PROGRAM prgAfterStationScan
VAR
END_VAR

//theme:ldUT4FLxql4
//call at the end of scan of stations..
//..for data to be processed after all values of a station
actAnyAlarmsGlobal();
actAnyWarningGlobal();

ACTION actAnyAlarmsGlobal:
//call for end of scan
//if any station has fault state, then set logic for all stations...
//writes to data multiple times due to manipulation of scan
IF 
	GlobalMessages.gMsgS1Stat.IsAlarm OR 
	GlobalMessages.gMsgS2Stat.IsAlarm OR 
	GlobalMessages.gMsgS3Stat.IsAlarm OR 
	GlobalMessages.gMsgS4Stat.IsAlarm OR 
	GlobalMessages.gMsgS5Stat.IsAlarm OR 
	GlobalMessages.gMsgS6Stat.IsAlarm OR
	GlobalMessages.gMsgMcStat.IsAlarm
THEN
	S1_Global.hmiHeader.AnyStationFaultHeaderActive := System.OneSecond;
	S2_Global.hmiHeader.AnyStationFaultHeaderActive := System.OneSecond;
	S3_Global.hmiHeader.AnyStationFaultHeaderActive := System.OneSecond;
	S4_Global.hmiHeader.AnyStationFaultHeaderActive := System.OneSecond;
	S5_Global.hmiHeader.AnyStationFaultHeaderActive := System.OneSecond;
	S6_Global.hmiHeader.AnyStationFaultHeaderActive := System.OneSecond;
	
	S1_Global.hmiHeader.AnyStationFaultColour		:= HMIColour.colourRed;
	S2_Global.hmiHeader.AnyStationFaultColour		:= HMIColour.colourRed;
	S3_Global.hmiHeader.AnyStationFaultColour		:= HMIColour.colourRed;
	S4_Global.hmiHeader.AnyStationFaultColour		:= HMIColour.colourRed;
	S5_Global.hmiHeader.AnyStationFaultColour		:= HMIColour.colourRed;
	S6_Global.hmiHeader.AnyStationFaultColour		:= HMIColour.colourRed;
	
	S1_Global.hmiHeader.isAnyFaultState				:= TRUE;
	S2_Global.hmiHeader.isAnyFaultState				:= TRUE;
	S3_Global.hmiHeader.isAnyFaultState				:= TRUE;
	S4_Global.hmiHeader.isAnyFaultState				:= TRUE;
	S5_Global.hmiHeader.isAnyFaultState				:= TRUE;
	S6_Global.hmiHeader.isAnyFaultState				:= TRUE;
	
ELSE
	S1_Global.hmiHeader.AnyStationFaultHeaderActive := FALSE;
	S2_Global.hmiHeader.AnyStationFaultHeaderActive := FALSE;
	S3_Global.hmiHeader.AnyStationFaultHeaderActive := FALSE;
	S4_Global.hmiHeader.AnyStationFaultHeaderActive := FALSE;
	S5_Global.hmiHeader.AnyStationFaultHeaderActive := FALSE;
	S6_Global.hmiHeader.AnyStationFaultHeaderActive := FALSE;

	S1_Global.hmiHeader.AnyStationFaultColour		:= HMIColour.colourBlue;
	S2_Global.hmiHeader.AnyStationFaultColour		:= HMIColour.colourBlue;
	S3_Global.hmiHeader.AnyStationFaultColour		:= HMIColour.colourBlue;
	S4_Global.hmiHeader.AnyStationFaultColour		:= HMIColour.colourBlue;
	S5_Global.hmiHeader.AnyStationFaultColour		:= HMIColour.colourBlue;
	S6_Global.hmiHeader.AnyStationFaultColour		:= HMIColour.colourBlue;

	S1_Global.hmiHeader.isAnyFaultState				:= FALSE;
	S2_Global.hmiHeader.isAnyFaultState				:= FALSE;
	S3_Global.hmiHeader.isAnyFaultState				:= FALSE;
	S4_Global.hmiHeader.isAnyFaultState				:= FALSE;
	S5_Global.hmiHeader.isAnyFaultState				:= FALSE;
	S6_Global.hmiHeader.isAnyFaultState				:= FALSE;	
END_IF

	//set indicators to 0
	S1_Global.hmiHeader.AnyStationFaultHeader := 0;
	S2_Global.hmiHeader.AnyStationFaultHeader := 0;
	S3_Global.hmiHeader.AnyStationFaultHeader := 0;
	S4_Global.hmiHeader.AnyStationFaultHeader := 0;
	S5_Global.hmiHeader.AnyStationFaultHeader := 0;
	S6_Global.hmiHeader.AnyStationFaultHeader := 0;

//write station 1 is in fault
IF 	S1_Global.hmiHeader.isFaultState THEN
	S1_Global.hmiHeader.AnyStationFaultHeader := 1;
	S2_Global.hmiHeader.AnyStationFaultHeader := 1;
	S3_Global.hmiHeader.AnyStationFaultHeader := 1;
	S4_Global.hmiHeader.AnyStationFaultHeader := 1;
	S5_Global.hmiHeader.AnyStationFaultHeader := 1;
	S6_Global.hmiHeader.AnyStationFaultHeader := 1;
END_IF

//write station 2 is in fault
IF 	S2_Global.hmiHeader.isFaultState THEN
	S1_Global.hmiHeader.AnyStationFaultHeader := 2;
	S2_Global.hmiHeader.AnyStationFaultHeader := 2;
	S3_Global.hmiHeader.AnyStationFaultHeader := 2;
	S4_Global.hmiHeader.AnyStationFaultHeader := 2;
	S5_Global.hmiHeader.AnyStationFaultHeader := 2;
	S6_Global.hmiHeader.AnyStationFaultHeader := 2;
END_IF

//write station 3 is in fault
IF 	S3_Global.hmiHeader.isFaultState THEN
	S1_Global.hmiHeader.AnyStationFaultHeader := 3;
	S2_Global.hmiHeader.AnyStationFaultHeader := 3;
	S3_Global.hmiHeader.AnyStationFaultHeader := 3;
	S4_Global.hmiHeader.AnyStationFaultHeader := 3;
	S5_Global.hmiHeader.AnyStationFaultHeader := 3;
	S6_Global.hmiHeader.AnyStationFaultHeader := 3;
END_IF

//write station 4 is in fault
IF 	S4_Global.hmiHeader.isFaultState THEN
	S1_Global.hmiHeader.AnyStationFaultHeader := 4;
	S2_Global.hmiHeader.AnyStationFaultHeader := 4;
	S3_Global.hmiHeader.AnyStationFaultHeader := 4;
	S4_Global.hmiHeader.AnyStationFaultHeader := 4;
	S5_Global.hmiHeader.AnyStationFaultHeader := 4;
	S6_Global.hmiHeader.AnyStationFaultHeader := 4;
END_IF

//write station 5 is in fault
IF 	S5_Global.hmiHeader.isFaultState THEN
	S1_Global.hmiHeader.AnyStationFaultHeader := 5;
	S2_Global.hmiHeader.AnyStationFaultHeader := 5;
	S3_Global.hmiHeader.AnyStationFaultHeader := 5;
	S4_Global.hmiHeader.AnyStationFaultHeader := 5;
	S5_Global.hmiHeader.AnyStationFaultHeader := 5;
	S6_Global.hmiHeader.AnyStationFaultHeader := 5;
END_IF

//write station 6 is in fault
IF 	S6_Global.hmiHeader.isFaultState THEN
	S1_Global.hmiHeader.AnyStationFaultHeader := 6;
	S2_Global.hmiHeader.AnyStationFaultHeader := 6;
	S3_Global.hmiHeader.AnyStationFaultHeader := 6;
	S4_Global.hmiHeader.AnyStationFaultHeader := 6;
	S5_Global.hmiHeader.AnyStationFaultHeader := 6;
	S6_Global.hmiHeader.AnyStationFaultHeader := 6;
END_IF

//..so it appears in all usage of the HMI for a given station

//add for base station header
IF GlobalMessages.gMsgMcStat.IsAlarm THEN
	//set special case for base machine
	S1_Global.hmiHeader.AnyStationFaultHeader := 99;
	S2_Global.hmiHeader.AnyStationFaultHeader := 99;
	S3_Global.hmiHeader.AnyStationFaultHeader := 99;
	S4_Global.hmiHeader.AnyStationFaultHeader := 99;
	S5_Global.hmiHeader.AnyStationFaultHeader := 99;
	S6_Global.hmiHeader.AnyStationFaultHeader := 99;
	
	S1_Global.hmiHeader.isFaultState := TRUE;
	S2_Global.hmiHeader.isFaultState := TRUE;
	S3_Global.hmiHeader.isFaultState := TRUE;
	S4_Global.hmiHeader.isFaultState := TRUE;
	S5_Global.hmiHeader.isFaultState := TRUE;
	S6_Global.hmiHeader.isFaultState := TRUE;
	
	S1_Global.hmiHeader.FaultStateHeader := 1;
	S2_Global.hmiHeader.FaultStateHeader := 1;
	S3_Global.hmiHeader.FaultStateHeader := 1;
	S4_Global.hmiHeader.FaultStateHeader := 1;
	S5_Global.hmiHeader.FaultStateHeader := 1;
	S6_Global.hmiHeader.FaultStateHeader := 1;
END_IF
END_ACTION

ACTION actAnyWarningGlobal:
//call for end of scan
//if any station has Warning state, then set logic for all stations...
//writes to data multiple times due to manipulation of scan
IF 
	GlobalMessages.gMsgS1Stat.IsWarning OR 
	GlobalMessages.gMsgS2Stat.IsWarning OR 
	GlobalMessages.gMsgS3Stat.IsWarning OR 
	GlobalMessages.gMsgS4Stat.IsWarning OR 
	GlobalMessages.gMsgS5Stat.IsWarning OR 
	GlobalMessages.gMsgS6Stat.IsWarning OR
	GlobalMessages.gMsgMcStat.IsWarning
THEN
	S1_Global.hmiHeader.AnyStationWarningHeaderActive := System.OneSecond;
	S2_Global.hmiHeader.AnyStationWarningHeaderActive := System.OneSecond;
	S3_Global.hmiHeader.AnyStationWarningHeaderActive := System.OneSecond;
	S4_Global.hmiHeader.AnyStationWarningHeaderActive := System.OneSecond;
	S5_Global.hmiHeader.AnyStationWarningHeaderActive := System.OneSecond;
	S6_Global.hmiHeader.AnyStationWarningHeaderActive := System.OneSecond;
	
	S1_Global.hmiHeader.AnyStationWarningColour		:= HMIColour.colourYellow;
	S2_Global.hmiHeader.AnyStationWarningColour		:= HMIColour.colourYellow;
	S3_Global.hmiHeader.AnyStationWarningColour		:= HMIColour.colourYellow;
	S4_Global.hmiHeader.AnyStationWarningColour		:= HMIColour.colourYellow;
	S5_Global.hmiHeader.AnyStationWarningColour		:= HMIColour.colourYellow;
	S6_Global.hmiHeader.AnyStationWarningColour		:= HMIColour.colourYellow;
	
	S1_Global.hmiHeader.isAnyWarningState				:= TRUE;
	S2_Global.hmiHeader.isAnyWarningState				:= TRUE;
	S3_Global.hmiHeader.isAnyWarningState				:= TRUE;
	S4_Global.hmiHeader.isAnyWarningState				:= TRUE;
	S5_Global.hmiHeader.isAnyWarningState				:= TRUE;
	S6_Global.hmiHeader.isAnyWarningState				:= TRUE;
	
ELSE
	S1_Global.hmiHeader.AnyStationWarningHeaderActive := FALSE;
	S2_Global.hmiHeader.AnyStationWarningHeaderActive := FALSE;
	S3_Global.hmiHeader.AnyStationWarningHeaderActive := FALSE;
	S4_Global.hmiHeader.AnyStationWarningHeaderActive := FALSE;
	S5_Global.hmiHeader.AnyStationWarningHeaderActive := FALSE;
	S6_Global.hmiHeader.AnyStationWarningHeaderActive := FALSE;

	S1_Global.hmiHeader.AnyStationWarningColour		:= HMIColour.colourBlue;
	S2_Global.hmiHeader.AnyStationWarningColour		:= HMIColour.colourBlue;
	S3_Global.hmiHeader.AnyStationWarningColour		:= HMIColour.colourBlue;
	S4_Global.hmiHeader.AnyStationWarningColour		:= HMIColour.colourBlue;
	S5_Global.hmiHeader.AnyStationWarningColour		:= HMIColour.colourBlue;
	S6_Global.hmiHeader.AnyStationWarningColour		:= HMIColour.colourBlue;

	S1_Global.hmiHeader.isAnyWarningState				:= FALSE;
	S2_Global.hmiHeader.isAnyWarningState				:= FALSE;
	S3_Global.hmiHeader.isAnyWarningState				:= FALSE;
	S4_Global.hmiHeader.isAnyWarningState				:= FALSE;
	S5_Global.hmiHeader.isAnyWarningState				:= FALSE;
	S6_Global.hmiHeader.isAnyWarningState				:= FALSE;	
END_IF

	//set indicators to 0
	S1_Global.hmiHeader.AnyStationWarningHeader := 0;
	S2_Global.hmiHeader.AnyStationWarningHeader := 0;
	S3_Global.hmiHeader.AnyStationWarningHeader := 0;
	S4_Global.hmiHeader.AnyStationWarningHeader := 0;
	S5_Global.hmiHeader.AnyStationWarningHeader := 0;
	S6_Global.hmiHeader.AnyStationWarningHeader := 0;

//write station 1 is in Warning
IF 	S1_Global.hmiHeader.isWarningState THEN
	S1_Global.hmiHeader.AnyStationWarningHeader := 1;
	S2_Global.hmiHeader.AnyStationWarningHeader := 1;
	S3_Global.hmiHeader.AnyStationWarningHeader := 1;
	S4_Global.hmiHeader.AnyStationWarningHeader := 1;
	S5_Global.hmiHeader.AnyStationWarningHeader := 1;
	S6_Global.hmiHeader.AnyStationWarningHeader := 1;
END_IF

//write station 2 is in Warning
IF 	S2_Global.hmiHeader.isWarningState THEN
	S1_Global.hmiHeader.AnyStationWarningHeader := 2;
	S2_Global.hmiHeader.AnyStationWarningHeader := 2;
	S3_Global.hmiHeader.AnyStationWarningHeader := 2;
	S4_Global.hmiHeader.AnyStationWarningHeader := 2;
	S5_Global.hmiHeader.AnyStationWarningHeader := 2;
	S6_Global.hmiHeader.AnyStationWarningHeader := 2;
END_IF

//write station 3 is in Warning
IF 	S3_Global.hmiHeader.isWarningState THEN
	S1_Global.hmiHeader.AnyStationWarningHeader := 3;
	S2_Global.hmiHeader.AnyStationWarningHeader := 3;
	S3_Global.hmiHeader.AnyStationWarningHeader := 3;
	S4_Global.hmiHeader.AnyStationWarningHeader := 3;
	S5_Global.hmiHeader.AnyStationWarningHeader := 3;
	S6_Global.hmiHeader.AnyStationWarningHeader := 3;
END_IF

//write station 4 is in Warning
IF 	S4_Global.hmiHeader.isWarningState THEN
	S1_Global.hmiHeader.AnyStationWarningHeader := 4;
	S2_Global.hmiHeader.AnyStationWarningHeader := 4;
	S3_Global.hmiHeader.AnyStationWarningHeader := 4;
	S4_Global.hmiHeader.AnyStationWarningHeader := 4;
	S5_Global.hmiHeader.AnyStationWarningHeader := 4;
	S6_Global.hmiHeader.AnyStationWarningHeader := 4;
END_IF

//write station 5 is in Warning
IF 	S5_Global.hmiHeader.isWarningState THEN
	S1_Global.hmiHeader.AnyStationWarningHeader := 5;
	S2_Global.hmiHeader.AnyStationWarningHeader := 5;
	S3_Global.hmiHeader.AnyStationWarningHeader := 5;
	S4_Global.hmiHeader.AnyStationWarningHeader := 5;
	S5_Global.hmiHeader.AnyStationWarningHeader := 5;
	S6_Global.hmiHeader.AnyStationWarningHeader := 5;
END_IF

//write station 6 is in Warning
IF 	S6_Global.hmiHeader.isWarningState THEN
	S1_Global.hmiHeader.AnyStationWarningHeader := 6;
	S2_Global.hmiHeader.AnyStationWarningHeader := 6;
	S3_Global.hmiHeader.AnyStationWarningHeader := 6;
	S4_Global.hmiHeader.AnyStationWarningHeader := 6;
	S5_Global.hmiHeader.AnyStationWarningHeader := 6;
	S6_Global.hmiHeader.AnyStationWarningHeader := 6;
END_IF

//..so it appears in all usage of the HMI for a given station

//add for base station header
IF GlobalMessages.gMsgMcStat.IsWarning THEN
	//set special case for base machine
	S1_Global.hmiHeader.AnyStationWarningHeader := 99;
	S2_Global.hmiHeader.AnyStationWarningHeader := 99;
	S3_Global.hmiHeader.AnyStationWarningHeader := 99;
	S4_Global.hmiHeader.AnyStationWarningHeader := 99;
	S5_Global.hmiHeader.AnyStationWarningHeader := 99;
	S6_Global.hmiHeader.AnyStationWarningHeader := 99;
	
	S1_Global.hmiHeader.isWarningState := TRUE;
	S2_Global.hmiHeader.isWarningState := TRUE;
	S3_Global.hmiHeader.isWarningState := TRUE;
	S4_Global.hmiHeader.isWarningState := TRUE;
	S5_Global.hmiHeader.isWarningState := TRUE;
	S6_Global.hmiHeader.isWarningState := TRUE;
	
	S1_Global.hmiHeader.WarningStateHeader := 1;
	S2_Global.hmiHeader.WarningStateHeader := 1;
	S3_Global.hmiHeader.WarningStateHeader := 1;
	S4_Global.hmiHeader.WarningStateHeader := 1;
	S5_Global.hmiHeader.WarningStateHeader := 1;
	S6_Global.hmiHeader.WarningStateHeader := 1;
END_IF
END_ACTION

END_PROGRAM

(* stored: Version 1.1.0.1, ProductVersion 3.1.4024.12
   POU prgAfterStationScan: Id {1a47d8fd-3e5d-4193-839a-5a5ee306ddc2}, SpecialFunc None
   Action actAnyAlarmsGlobal: Id {976dde39-5720-4a2c-860b-750f4fc28559}
   Action actAnyWarningGlobal: Id {a977cc66-8f5a-446a-96fb-20ddf805ab2d} *)
